# EPICS autosave request: NDFileEDF_settings.req
file "NDPluginFile_settings.req", P=$(P), R=$(R)
$(P)$(R)MinHeaderSize
